// TIA Portal V20 export
TYPE "typeSequenceControlNode_topTapeFixStage"
// stored: Namespace Unit1.Em3
   STRUCT
      jobs : "LAF_typeJobs";
      sequence : "LAF_typeSequence";
      selectJobStatus { S7_SetPoint := 'True'} : Array[0..10] of "LAF_typeJobStatus";
      "step" : "LER_typeStep";
      jobInterface : "Unit1.Em3.typeSequenceControlNodeJobInterface_topTapeFixStage";
      homeCheck : "Unit1.Em3.typeSequenceControlNodeHomeCheck_topTapeFixStage";
   END_STRUCT;
   // // "step".action1[101] : Step[101] : JOB[1] Condition
   // // "step".action1[110] : Step[110] : Top Tape Fix Stage Left/Center/Right Top Clamp Up
   // // "step".action1[111] : Step[111] : Top Tape Fix Stage Bottom Clamp Down
   // // "step".action1[120] : Step[120] : Top Tape Fix Stage Bottom Clamp Up
   // // "step".action1[121] : Step[121] : Top Tape Fix Stage Left/Center/Right Top Clamp Down
   // // "step".action1[180] : Step[180] : Top Tape Y-Axis Wait Pos
   // // "step".action1[190] : Step[190] : JOB[1] Step End
   // // "step".action1[201] : Step[201] : JOB[2] Condition
   // // "step".action1[210] : Step[210] : Top Tape Fix Stage [Loading Request] => JR PP Left
   // // "step".action1[220] : Step[220] Top Tape Y-Axis JR Put/Get Pos
   // // "step".action1[230] : Step[230] : Top Tape Fix Stage Bottom Clamp Up
   // // "step".action1[231] : Step[231] : Top Tape Fix Stage Left/Center/Right Top Clamp Down
   // // "step".action1[232] : Step[232] : Top Tape Fix Stage [Unclamp Request] => JR PP Left
   // // "step".action1[270] : Step[270] : Spare
   // // "step".action1[280] : Step[280] : Top Tape Y-Axis Wait Pos
   // // "step".action1[290] : Step[290] : JOB[2] Step End
   // // "step".action1[301] : Step[301] : JOB[3] Conditiion
   // // "step".action1[310] : Step[310] : Top Tape Fix Stage => Call Attachment Tape-1
   // // "step".action1[320] : Step[320] : Spare
   // // "step".action1[390] : Step[390] : JOB[3] Step End
   // // "step".action1[401] : Step[401] : JOB[4] Conditiion
   // // "step".action1[410] : Step[410] : Top Tape Fix Stage => Call Attachment Tape-1
   // // "step".action1[420] : Step[420] : Spare
   // // "step".action1[490] : Step[490] : JOB[4] Step End
   // // "step".action1[501] : Step[501] : JOB[5] Condition
   // // "step".action1[510] : Step[510] : Top Tape Fix Stage [Unloading Request] => JR PP Right
   // // "step".action1[520] : Step[520] : Top Tape Fix Stage Y-Axis Put/Get Pos
   // // "step".action1[530] : Step[530] : Top Tape Fix Stage [Clamp Request] => JR PP Right
   // // "step".action1[531] : Step[531] : Top Tape Fix Stage Left/Center/Right Top Clamp Up
   // // "step".action1[532] : Step[532] : Top Tape Fix Stage Bottom Clamp Down
   // // "step".action1[570] : Step[570] : Spare
   // // "step".action1[580] : Step[580] : Top Tape Y-Axis Wait Pos
   // // "step".action1[590] : Step[590] : JOB[5] Step End
   // // "step".transition1[101] : Step[101] : JOB[1] Condition
   // // "step".transition1[110] : Step[110] : Top Tape Fix Stage Left/Center/Right Top Clamp Up
   // // "step".transition1[111] : Step[111] : Top Tape Fix Stage Bottom Clamp Down
   // // "step".transition1[120] : Step[120] : Top Tape Fix Stage Bottom Clamp Up
   // // "step".transition1[121] : Step[121] : Top Tape Fix Stage Left/Center/Right Top Clamp Down
   // // "step".transition1[180] : Step[180] : Top Tape Y-Axis Wait Pos
   // // "step".transition1[190] : Step[190] : JOB[1] Step End
   // // "step".transition1[201] : Step[201] : JOB[2] Condition
   // // "step".transition1[210] : Step[210] : Top Tape Fix Stage [Loading Request] => JR PP Left
   // // "step".transition1[220] : Step[220] Top Tape Y-Axis JR Put/Get Pos
   // // "step".transition1[230] : Step[230] : Top Tape Fix Stage Bottom Clamp Up
   // // "step".transition1[231] : Step[231] : Top Tape Fix Stage Left/Center/Right Top Clamp Down
   // // "step".transition1[232] : Step[232] : Top Tape Fix Stage [Unclamp Request] => JR PP Left
   // // "step".transition1[270] : Step[270] : Spare
   // // "step".transition1[280] : Step[280] : Top Tape Y-Axis Wait Pos
   // // "step".transition1[290] : Step[290] : JOB[2] Step End
   // // "step".transition1[301] : Step[301] : JOB[3] Conditiion
   // // "step".transition1[310] : Step[310] : Top Tape Fix Stage => Call Attachment Tape-1
   // // "step".transition1[320] : Step[320] : Spare
   // // "step".transition1[390] : Step[390] : JOB[3] Step End
   // // "step".transition1[401] : Step[401] : JOB[4] Conditiion
   // // "step".transition1[410] : Step[410] : Top Tape Fix Stage => Call Attachment Tape-1
   // // "step".transition1[420] : Step[420] : Spare
   // // "step".transition1[490] : Step[490] : JOB[4] Step End
   // // "step".transition1[501] : Step[501] : JOB[5] Condition
   // // "step".transition1[510] : Step[510] : Top Tape Fix Stage [Unloading Request] => JR PP Right
   // // "step".transition1[520] : Step[520] : Top Tape Fix Stage Y-Axis Put/Get Pos
   // // "step".transition1[530] : Step[530] : Top Tape Fix Stage [Clamp Request] => JR PP Right
   // // "step".transition1[531] : Step[531] : Top Tape Fix Stage Left/Center/Right Top Clamp Up
   // // "step".transition1[532] : Step[532] : Top Tape Fix Stage Bottom Clamp Down
   // // "step".transition1[570] : Step[570] : Spare
   // // "step".transition1[580] : Step[580] : Top Tape Y-Axis Wait Pos
   // // "step".transition1[590] : Step[590] : JOB[5] Step End
END_TYPE
